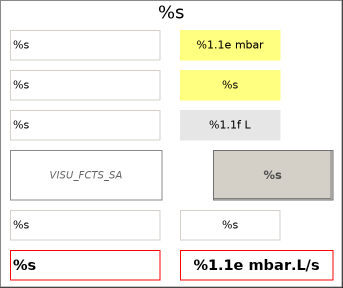
VISUALIZATION SA_TEST_RP  // 343x288
VAR_IN_OUT
	m_Input_Operation:		BLOCK_OPERATION;
	m_Input_Pression:		REAL;		(*PRM pression initiale*)
	m_Input_Duree:			TIME;		(*PRM temps du test*)
	m_Input_Volume:			REAL;		(*CONF volume*)
	m_Input_Co_Stop:		BOOL;		(*Co stop*)
	m_Input_Timer:			TIME;		(*Tps écoulé*)
	m_Input_Result:			REAL;		(*Résultat*)
END_VAR
    Rectangle (0,0 343x288), "%s", text list: 'TextList_Test_RP', text index: 0
    Textfield (10,30 150x30), "%s", text list: 'TextList_Test_RP', text index: 1
    Textfield (10,70 150x30), "%s", text list: 'TextList_Test_RP', text index: 2
    Textfield (10,110 150x30), "%s", text list: 'TextList_Test_RP', text index: 3
    Textfield (10,210 150x30), "%s", invisible if: m_Input_Operation.OK OR m_Input_Operation.AR, text list: 'TextList_Test_RP', text index: 4
    Textfield (10,250 150x30), "%s", invisible if: m_Input_Operation.EC, text list: 'TextList_Test_RP', text index: 5
    Textfield (180,30 100x30), "%1.1e mbar", text variable: m_Input_Pression, input disabled if: (NOT PRG_USER.ACTU_USER.FONCTION_SA AND NOT MACHINE.STATE_Prod) OR MACHINE.STATE_Prod
        OnMouseClick: write the text variable via InputWithLimits, min 0, max 1000
    Textfield (180,70 100x30), "%s", text variable: m_Input_Duree, input disabled if: (NOT PRG_USER.ACTU_USER.FONCTION_SA AND NOT MACHINE.STATE_Prod) OR MACHINE.STATE_Prod
        OnMouseClick: write the text variable via InputWithLimits
    Textfield (180,110 100x30), "%1.1f L", text variable: m_Input_Volume
    Frame (10,150 152x50)
        shows VISU_FCTS_SA(m_Input_ID_XML := 5, m_Input_UserRight := PRG_USER.ACTU_USER.FONCTION_SA AND NOT MACHINE.STATE_PROD, m_Input_Operation := m_Input_Operation)
    Button (213,150 120x50), "%s", input disabled if: NOT (PRG_User.ACTU_USER.FONCTION_SA AND NOT MACHINE.STATE_PROD), text list: 'TextList_Test_RP', text index: 6
        toggle m_Input_Co_Stop
    Textfield (180,210 100x30), "%s", text variable: m_Input_Timer, invisible if: m_Input_Operation.OK OR m_Input_Operation.AR
    Textfield (180,250 153x30), "%1.1e mbar.L/s", text variable: m_Input_Result, invisible if: m_Input_Operation.EC
END_VISUALIZATION

(* stored: Version 1.1.0.1, ProductVersion 3.1.4024.12
   Visu SA_TEST_RP: Id {9c4c2f61-bb4b-4bfe-bb86-c092183ea13b} *)
